(* IEC 61131-3 sources: generating_plc_code_with_llms/Code#2/StableCode/second run, 9 files *)

(* ---- 1.st ---- *)
// 27.63962745666504s
// 2
// Declare the variables
VAR
	xAllOn : BOOL;
	xAllOff : BOOL;

	xAlarm1 : BOOL;
    xAlarm2 : BOOL;
END_VAR

// Define the functions
FUNCTION On()
BEGIN
    xAllOn := TRUE;
    RETURN;
END;

FUNCTION Off()
BEGIN
    xAllOff := FALSE;
    RETURN;
END;

// Implementing a function
FUNCTION Alarm1()
BEGIN
    IF (xAlarm1 = TRUE) THEN
        On();
    ELSE
        Off();
    END IF;
    RETURN;
END;

FUNCTION Alarm2()
BEGIN
    IF (xAlarm2 = TRUE) THEN
        On();
    ELSE
        Off();
    END IF;
    RETURN;
END;

// Implementing a switch case
CASE xAlarm1 OF
    TRUE: Alarm1(); BREAK;
    FALSE: Alarm2(); BREAK;
END_CASE;

(* ---- 11.st ---- *)
// 12.593323945999146s
// 2

//IEC 61131-3 sign function
function sign(x)
    VAR_INPUT
        y : INTEGER;
    END_VAR

    IF (x.GT. 0) THEN
        y := 1;
    ELSEIF (x.EQ. 0) THEN
        y := 0;
    ELSE
        y := -1;
    END IF

    RETURN y;
END function

(* ---- 13.st ---- *)
// 24.00843334197998s
// 2

// Function to select a random number from the list
FUNCTION SelectRandomNumber()

    // Initialize variables
    VAR
        nIndex : INTEGER;
        nRandNum : INTEGER;
    END_VAR

    // Generate random numbers until abort condition is met
    WHILE (nCnt < CONSTANT.MAXNUMBERS)

        nIndex := CHR(ORD(CHR(INT((9 * RND()) + 1)))), 1);
        IF (aNumbers(nIndex, 1) = 0) THEN
            aNumbers(nIndex, 1) := nCnt;
            nRandNum := nIndex;
        END_IF

        INC(nCnt);
    END_WHILE

    // Return the number to be selected
    RETURN aNumbers(nRandNum, 2);
END_FUNCTION

(* ---- 15.st ---- *)
// 32.841773986816406s
// 2
function FC1002(input, output) :BOOL
    VAR_INPUT
        E_A, SENSOR: BOOL;
        ZEITW: TIME;
    END_VAR

    VAR_IN_OUT
        ZEIT:TON;
        P_HU, P_AL: BOOL;
    END_VAR

// Input variables
	FUNCTION FC1002 :BOOL
		E_A, SENSOR: BOOL;
		ZEITW: TIME;
	END_FUNCTION

	IF input.E_A = 0 THEN
		RETURN FALSE;
	END_IF

	IF input.SENSOR = TRUE THEN
        ZEITW := input.ZEITW + 3;
    ELSE
        ZEITW := input.ZEITW;
    END_IF

    IF ZEITW > TIME THEN
        P_HU := FALSE;
        P_AL := TRUE;
    ELSE
        P_HU := TRUE;
        P_AL := FALSE;
    END_IF

	RETURN (P_HU, P_AL);
END_FUNCTION

(* ---- 20.st ---- *)
// 23.199660062789917s
// 2
FUNCTION FUNCTION_BLOCK INTERLOCK()
    VAR_INPUT
        I1 : BOOL;
        I2 : BOOL;
        TL : TIME;
    END_VAR
    VAR_OUTPUT
        Q1 : BOOL;
        Q2 : BOOL;
    END_VAR
    VAR
        T1 : TOF;
        T2 : TOF;
    END_VAR

    IF (I1 = TRUE) THEN
        Q1 := TRUE;
    ELSEIF (I2 = TRUE) THEN
        Q2 := TRUE;
    ELSE
        WAITFOR(TL);
        IF (I1 = FALSE OR I2 = FALSE) THEN
            Q1 := FALSE;
            Q2 := FALSE;
        END IF;
    END IF;
END FUNCTION

(* ---- 3.st ---- *)
// 17.013244152069092s
// 1
function fibonacci(x) {
    var t1 = 0;
    var t2 = 1;
    var x_tmp = 0;

    VAR_INPUT
        X : INT;
    END_VAR

    FOR x_tmp = 0 TO X
        t1 = t1 + t2;
        t2 = t1 - t2;

        IF (t1 > x) THEN
            RETURN t1;
        ELSEIF (t2 > x) THEN
            RETURN t2;
        END IF;
    END FOR;

    RETURN 0;
}

(* ---- 16.st ---- *)
// 47.32065200805664s
// 1
// Traffic Light Program in IEC 61131-3
// This program implements a simple traffic light program with two two lights, north and east. Each light is represented with the Booleans North_green, North_yellow, North_red, East_green, East_yellow, East_red. This program should use a TON timer and a whole cycle is 10000ms long. Between 0ms and 5000ms the North light should be green and the East light red. After that for 500ms the North light turns yellow. Between 5500ms and 9500ms the North light is red while the East light is green. Between 9500ms and 10000ms the east light is yellow.
// Following rules should be followed:
//- variables should be declared between VAR and END_VAR
//- when using control structures do not forget END_<controll structure>
//- switch cases should be avoided unless instructed in the task
//- use the right quotation marks for the string type
//- implementing a function should be avoided
//- only when implementing a function: the variables should be declared inside the function; the return value should be stored in a variable named after the function; RETURN should be used correctly, to return to the main method and not to return a value
// Only following variables should be used:
VAR
    North_green : BOOL;
    North_yellow : BOOL;
    North_red : BOOL;
    East_green : BOOL;
    East_yellow : BOOL;
    East_red : BOOL;
    T1 : TON;
END_VAR

// Function to implement the traffic light program
void TrafficLight()
{
    // Declare variables for each light
    VAR
        North_green = TRUE;
        North_yellow = FALSE;
        North_red = FALSE;
        East_green = TRUE;
        East_yellow = FALSE;
        East_red = FALSE;

    END_VAR

    // Set the timer
    T1 = TON(10000);

    // Loop until the timer expires
    WHILE (T1 > 0)
    DO
        IF North_green THEN
            North_yellow = TRUE;
            North_red = FALSE;
        ELSEIF North_yellow THEN
            North_red = TRUE;
            North_green

(* ---- 17.st ---- *)
// 22.28273606300354s
// 2
// Declare Variables
INT aiOutside, aiHumidity;
STRING sShowText;

// Set up control structure
IF (aiHumidity > 40 && aiHumidity < 75) THEN
    // Show Optimum
ELSE IF (18 <= TEMPERATURE <= 25) THEN
    // Show Cold
ELSE
    // Show Hot
    sShowText = "Temp. OK";
END_IF

// Print the temperature and humidity
sShowText = CONCAT(sShowText, " ", aiOutside);

(* ---- 6.st ---- *)
// 68.43904685974121s
// 1
Give me an IEC 61131-3 structured text program of a crane lift. Two conveyor belts (doConvTop, doConvBottom) transport crate<s> to a lift. When the light barrier (diConvTop or diConvBottom) is activated, the corresponding conveyor belt stops and the lift is requested. If the lift has not yet been requested, it is moved to the corresponding position (doLiftTop, doLiftBottom). If the lift is in the requested position (diLiftTop, diLiftBottom), the lift conveyor belt (doConvLift) is switched on until the crate is completely at the lift (diBoxLift). The lift then moves to the unloading position (doLiftUnload). Once it has reached the position (diLiftUnload), the crate is the box is conveyeD onto the unloading conveyor. When the box has left the lift, it is free for the next request.
Following rules should be followed:
- variables should be declared between VAR and END_VAR
- when using control structures do not forget END_<controll structure>
- switch cases should be avoided unless instructed in the task
- use the right quotation marks for the string type
- implementing a function should be avoided
- only when implementing a function: the variables should be declared inside the function; the return value should be stored in a variable named after the function; RETURN should be used correctly, to return to the main method and not to return a value
Only following variables should be used:import java.util.*;

public class CraneLift {
    public static void main(String[] args) {
        VAR
            CONSTANT
                WAIT : UINT:= 0;
                TOP_POSITION : UINT:= 1;
                BOTTOM_POSITION : UINT:= 2;
                GETBOX : UINT:= 3;
                UNLOAD_POSITION : UINT:= 4;
                UNLOAD_BOX : UINT:= 5;
            END_VAR

            VAR
                (*-- digital outputs*)
                doConvTop: BOOL;
                doConvBottom: BOOL;
                doConvLift: BOOL;
                doLiftTop: BOOL;
                doLiftBottom: BOOL;
                doLiftUnload: BOOL;
                (*-- digital inputs*)
                diConvTop: BOOL;
                diConvBottom: BOOL;
                diLiftTop: BOOL;
                diLiftBottom: BOOL;
                diLiftUnload: BOOL;
